// TIA Portal V20 export
FUNCTION_BLOCK "LER_RadiusMeasure"   // FB121, LAD
// stored: Access Published, MemoryReserve 100, SetENOAutomatically false
   VAR_INPUT
      enable : Bool;
      enableManualCmds : Bool;
      radiusProcessValue : LReal;
   END_VAR
   VAR_OUTPUT
      ProcessValueZeroSet : LReal;
      radius : LReal;
      diameter : LReal;
   END_VAR
   VAR_IN_OUT
      configruation : "LER_typeRadiusMeasureConfiguration";
      moduleInterface : "LER_typeRadiusMeasureInterface";
      controlNode : "LER_typeRadiusMeasureControlNode";
   END_VAR
   VAR RETAIN
      statRadiusProcessValueZeroSetOffset : LReal;
   END_VAR
   VAR
      statRadiusProcessValueBuffer : Array[0..5] of LReal;
      statOffset : LReal;
   END_VAR
   VAR_TEMP
      P_TRIG : Array[0..10] of Bool;
   END_VAR
   VAR_TEMP   // added for the SCL form of the ladder/FBD networks
      _w1 : Bool;
      _w2 : Bool;
      _w3 : Bool;
   END_VAR
BEGIN

REGION Network 1: Radius Process Value ZeroSet
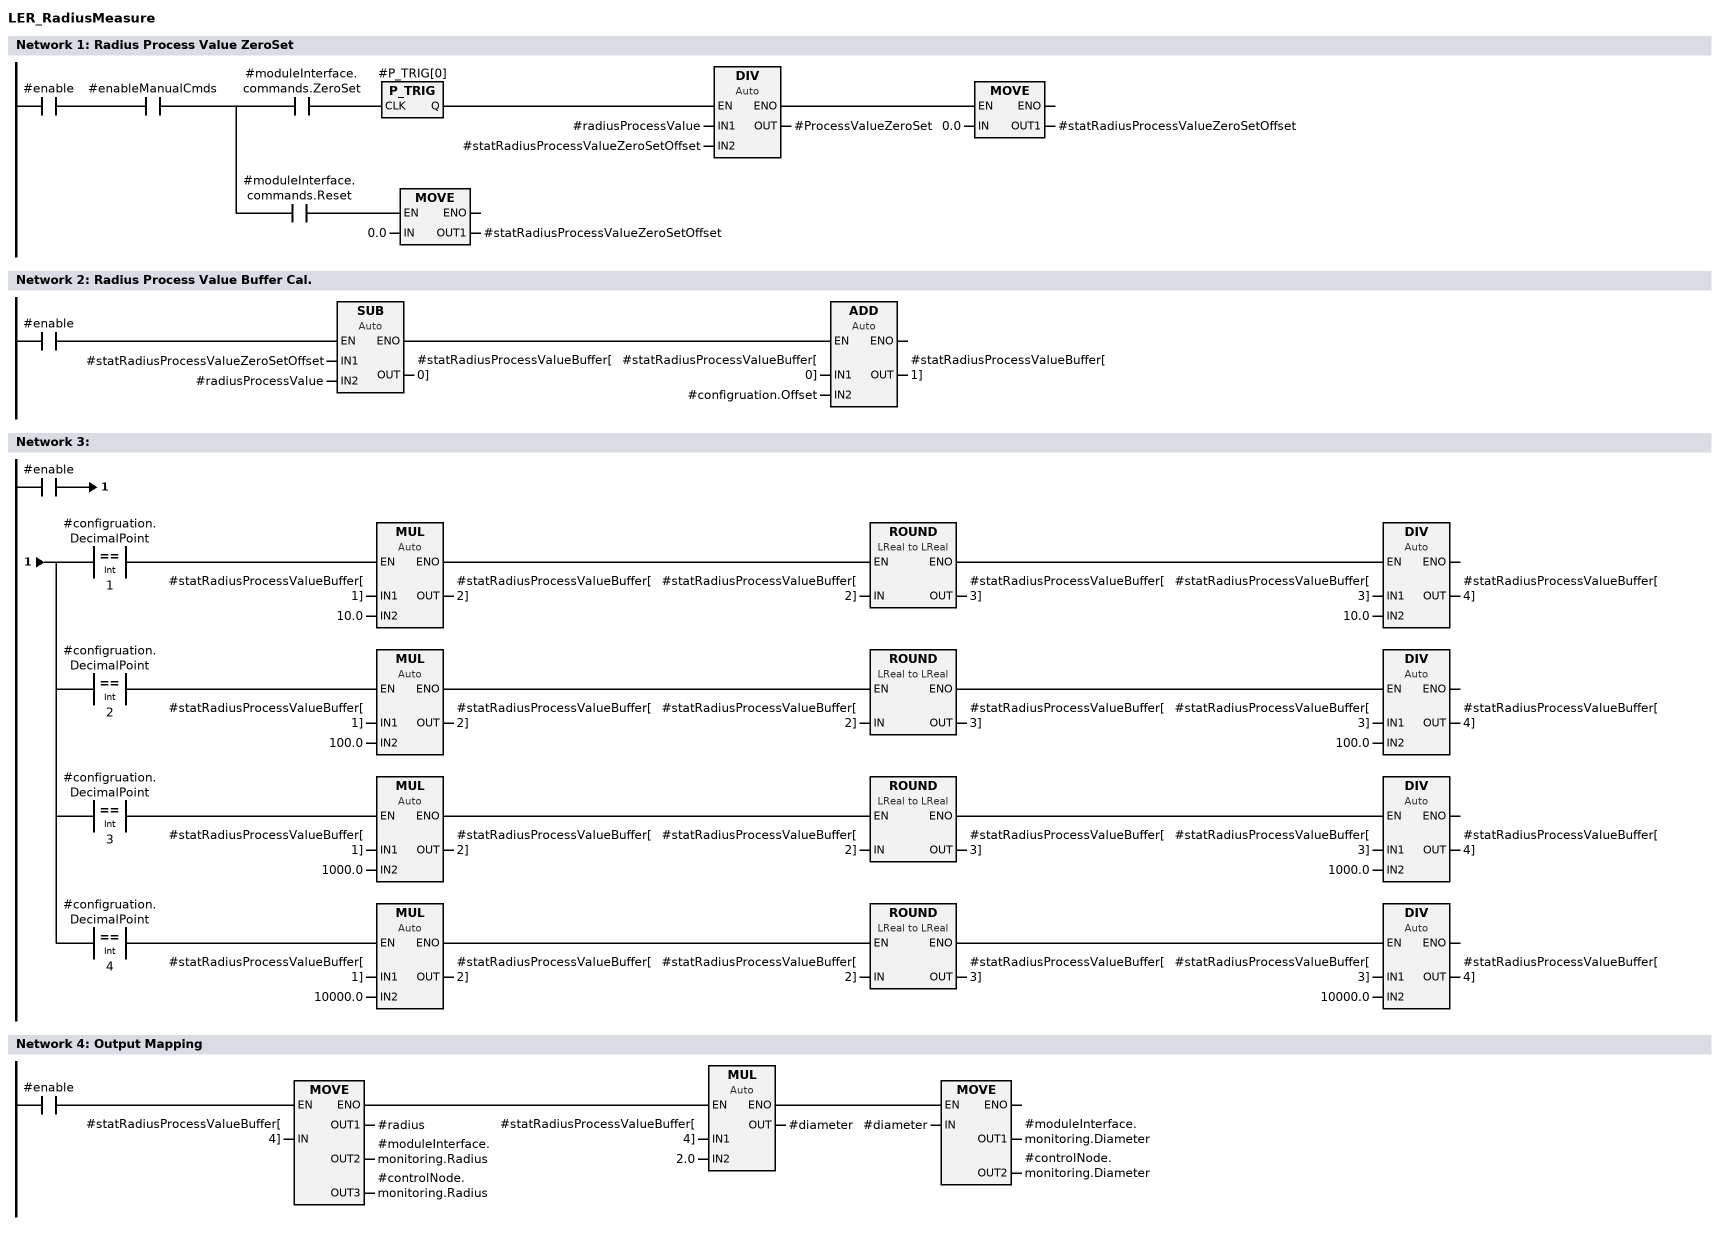
   RUNG wire#powerrail
      Contact( #enable )
      Contact( #enableManualCmds )
      wire#w1
      Contact( #moduleInterface.commands.ZeroSet )
      P_Trig( #P_TRIG[0] )
      Div(in1 := #radiusProcessValue, in2 := #statRadiusProcessValueZeroSetOffset, out => #ProcessValueZeroSet)
      Move(in := 0.0, out1 => #statRadiusProcessValueZeroSetOffset)
   END_RUNG
   RUNG wire#w1
      Contact( #moduleInterface.commands.Reset )
      Move(in := 0.0, out1 => #statRadiusProcessValueZeroSetOffset)
   END_RUNG
   // the same network as SCL:
   #_w1 := #enable AND #enableManualCmds;
   #_w2 := #_w1 AND #moduleInterface.commands.ZeroSet;
   #_w3 := #_w2 AND NOT #P_TRIG[0];   // rising edge
   #P_TRIG[0] := #_w2;
   IF #_w3 THEN
       #ProcessValueZeroSet := #radiusProcessValue / #statRadiusProcessValueZeroSetOffset;
       #statRadiusProcessValueZeroSetOffset := 0.0;
   END_IF;
   IF #_w1 AND #moduleInterface.commands.Reset THEN #statRadiusProcessValueZeroSetOffset := 0.0; END_IF;
END_REGION

REGION Network 2: Radius Process Value Buffer Cal.
   RUNG wire#powerrail
      Contact( #enable )
      Sub(in1 := #statRadiusProcessValueZeroSetOffset, in2 := #radiusProcessValue, out => #statRadiusProcessValueBuffer[0])
      Add(in1 := #statRadiusProcessValueBuffer[0], in2 := #configruation.Offset, out => #statRadiusProcessValueBuffer[1])
   END_RUNG
   // the same network as SCL:
   IF #enable THEN
       #statRadiusProcessValueBuffer[0] := #statRadiusProcessValueZeroSetOffset - #radiusProcessValue;
       #statRadiusProcessValueBuffer[1] := #statRadiusProcessValueBuffer[0] + #configruation.Offset;
   END_IF;
END_REGION

REGION Network 3
   RUNG wire#powerrail
      Contact( #enable )
      wire#w1
      { S7_Templates := "SrcType := Int" } EQ_Contact(in1 := #configruation.DecimalPoint, in2 := 1)
      Mul(in1 := #statRadiusProcessValueBuffer[1], in2 := 10.0, out => #statRadiusProcessValueBuffer[2])
      { S7_Templates := "[SrcType := LReal, DestType := LReal]" } Round(in := #statRadiusProcessValueBuffer[2], out => #statRadiusProcessValueBuffer[3])
      Div(in1 := #statRadiusProcessValueBuffer[3], in2 := 10.0, out => #statRadiusProcessValueBuffer[4])
   END_RUNG
   RUNG wire#w1
      { S7_Templates := "SrcType := Int" } EQ_Contact(in1 := #configruation.DecimalPoint, in2 := 2)
      Mul(in1 := #statRadiusProcessValueBuffer[1], in2 := 100.0, out => #statRadiusProcessValueBuffer[2])
      { S7_Templates := "[SrcType := LReal, DestType := LReal]" } Round(in := #statRadiusProcessValueBuffer[2], out => #statRadiusProcessValueBuffer[3])
      Div(in1 := #statRadiusProcessValueBuffer[3], in2 := 100.0, out => #statRadiusProcessValueBuffer[4])
   END_RUNG
   RUNG wire#w1
      { S7_Templates := "SrcType := Int" } EQ_Contact(in1 := #configruation.DecimalPoint, in2 := 3)
      Mul(in1 := #statRadiusProcessValueBuffer[1], in2 := 1000.0, out => #statRadiusProcessValueBuffer[2])
      { S7_Templates := "[SrcType := LReal, DestType := LReal]" } Round(in := #statRadiusProcessValueBuffer[2], out => #statRadiusProcessValueBuffer[3])
      Div(in1 := #statRadiusProcessValueBuffer[3], in2 := 1000.0, out => #statRadiusProcessValueBuffer[4])
   END_RUNG
   RUNG wire#w1
      { S7_Templates := "SrcType := Int" } EQ_Contact(in1 := #configruation.DecimalPoint, in2 := 4)
      Mul(in1 := #statRadiusProcessValueBuffer[1], in2 := 10000.0, out => #statRadiusProcessValueBuffer[2])
      { S7_Templates := "[SrcType := LReal, DestType := LReal]" } Round(in := #statRadiusProcessValueBuffer[2], out => #statRadiusProcessValueBuffer[3])
      Div(in1 := #statRadiusProcessValueBuffer[3], in2 := 10000.0, out => #statRadiusProcessValueBuffer[4])
   END_RUNG
   // the same network as SCL:
   IF #enable AND (#configruation.DecimalPoint = 1) THEN
       #statRadiusProcessValueBuffer[2] := #statRadiusProcessValueBuffer[1] * 10.0;
       #statRadiusProcessValueBuffer[3] := ROUND(#statRadiusProcessValueBuffer[2]);
       #statRadiusProcessValueBuffer[4] := #statRadiusProcessValueBuffer[3] / 10.0;
   END_IF;
   IF #enable AND (#configruation.DecimalPoint = 2) THEN
       #statRadiusProcessValueBuffer[2] := #statRadiusProcessValueBuffer[1] * 100.0;
       #statRadiusProcessValueBuffer[3] := ROUND(#statRadiusProcessValueBuffer[2]);
       #statRadiusProcessValueBuffer[4] := #statRadiusProcessValueBuffer[3] / 100.0;
   END_IF;
   IF #enable AND (#configruation.DecimalPoint = 3) THEN
       #statRadiusProcessValueBuffer[2] := #statRadiusProcessValueBuffer[1] * 1000.0;
       #statRadiusProcessValueBuffer[3] := ROUND(#statRadiusProcessValueBuffer[2]);
       #statRadiusProcessValueBuffer[4] := #statRadiusProcessValueBuffer[3] / 1000.0;
   END_IF;
   IF #enable AND (#configruation.DecimalPoint = 4) THEN
       #statRadiusProcessValueBuffer[2] := #statRadiusProcessValueBuffer[1] * 10000.0;
       #statRadiusProcessValueBuffer[3] := ROUND(#statRadiusProcessValueBuffer[2]);
       #statRadiusProcessValueBuffer[4] := #statRadiusProcessValueBuffer[3] / 10000.0;
   END_IF;
END_REGION

REGION Network 4: Output Mapping
   RUNG wire#powerrail
      Contact( #enable )
      Move(in := #statRadiusProcessValueBuffer[4], out1 => #radius, out2 => #moduleInterface.monitoring.Radius, out3 => #controlNode.monitoring.Radius)
      Mul(in1 := #statRadiusProcessValueBuffer[4], in2 := 2.0, out => #diameter)
      Move(in := #diameter, out1 => #moduleInterface.monitoring.Diameter, out2 => #controlNode.monitoring.Diameter)
   END_RUNG
   // the same network as SCL:
   IF #enable THEN
       #radius := #statRadiusProcessValueBuffer[4];
       #moduleInterface.monitoring.Radius := #statRadiusProcessValueBuffer[4];
       #controlNode.monitoring.Radius := #statRadiusProcessValueBuffer[4];
       #diameter := #statRadiusProcessValueBuffer[4] * 2.0;
       #moduleInterface.monitoring.Diameter := #diameter;
       #controlNode.monitoring.Diameter := #diameter;
   END_IF;
END_REGION
END_FUNCTION_BLOCK
